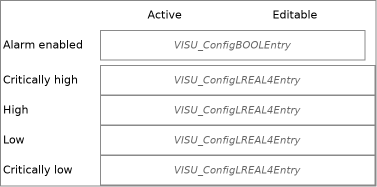
VISUALIZATION VISU_HiHiLoLoAlarmConfig  // 377x187
VAR_IN_OUT
	active : HiHiLoLoAlarmConfig;
    editable : HiHiLoLoAlarmConfig;
END_VAR
    Label (0,30 135x30), "Alarm enabled"
    Frame (100,30 265x30)
        shows VISU_ConfigBOOLEntry(active := active.enabled, editable := editable.enabled)
    Label (0,65 105x30), "Critically high"
    Frame (100,65 275x30)
        shows VISU_ConfigLREAL4Entry(active := active.hiHi, editable := editable.hiHi)
    Label (0,95 105x30), "High"
    Frame (100,95 275x30)
        shows VISU_ConfigLREAL4Entry(active := active.hi, editable := editable.hi)
    Label (0,125 105x30), "Low"
    Frame (100,125 275x30)
        shows VISU_ConfigLREAL4Entry(active := active.lo, editable := editable.lo)
    Label (0,155 105x30), "Critically low"
    Frame (100,155 275x30)
        shows VISU_ConfigLREAL4Entry(active := active.loLo, editable := editable.loLo)
    Label (100,0 130x30), "Active"
    Label (230,0 130x30), "Editable"
END_VISUALIZATION

(* stored: Version 1.1.0.1, ProductVersion 3.1.4019.2
   Visu VISU_HiHiLoLoAlarmConfig: Id {a5d5296d-43e6-4f7b-8196-c5cd382816fb} *)
